INTERFACE I_MessageData

PROPERTY DirRoot : POINTER to string(255)
SET
END_SET
END_PROPERTY

PROPERTY ErrorIndex : reference to uint
SET
END_SET
END_PROPERTY

PROPERTY FileRoot : pointer to string(255)
SET
END_SET
END_PROPERTY

PROPERTY LocalTime : pointer to DT
SET
END_SET
END_PROPERTY

PROPERTY MessageIndex : reference to uint
SET
END_SET
END_PROPERTY

PROPERTY MsgList : pointer to ARRAY[1..GVL_MSG.MAX_MESSAGE] OF st_message
SET
END_SET
END_PROPERTY

END_INTERFACE

(* stored: Version 1.1.0.1, ProductVersion 3.1.4026.13
   Itf I_MessageData: Id {e76eb09d-fc94-4cb1-bb48-a200667ba7e5}
   Property DirRoot: Id {83fe4674-1a2e-48c9-ba35-5e14525c70e5}
   Set Set: Id {a24f4d7b-65e2-472e-ad0f-85df0cab56fa}
   Property ErrorIndex: Id {8594822f-fb8f-4b71-86af-5c219592b0b0}
   Set Set: Id {81c11735-0851-4a3d-8929-f734c5145f2d}
   Property FileRoot: Id {99cdb962-29bf-4e9f-b4b0-94875e78da4d}
   Set Set: Id {2aee7dc8-9eab-4432-add5-056d1799f72e}
   Property LocalTime: Id {ec8eb63d-cd43-4261-8d8e-a627dae210d7}
   Set Set: Id {0b9c1a02-780e-42e7-a8b9-f0437d3c675c}
   Property MessageIndex: Id {cabeeaaf-b2d0-4544-8a8f-c462bfcc4635}
   Set Set: Id {7a046084-3acc-4b49-8605-8e155573405d}
   Property MsgList: Id {2875394a-25ed-4476-afc6-3f73bf082a6f}
   Set Set: Id {fa0095c1-7189-4d24-b7ae-abb626fbd6a8} *)
